FUNCTION_BLOCK FB_mF EXTENDS FB_StateSpaceModel
VAR_INPUT
END_VAR
VAR_OUTPUT
END_VAR
VAR
END_VAR

METHOD PUBLIC Init
VAR_INPUT
	activateObserver : BOOL;
END_VAR
VAR
    i,j : INT;
END_VAR

SUPER^();
nx := 2;
nu := 2;
ny := 1;

// Load matrices
_A[1,1] := 0.9895;
_A[1,2] := 0.03677;
_A[2,1] := -0.01237;
_A[2,2] := 0.9649;

_B[1,1] := -2.52E-05;
_B[1,2] := -1.673E-06;
_B[2,1] := -2.199E-04;
_B[2,2] := -5.346E-06;

_C[1,1] := -10.22;
_C[1,2] := -0.1235;

_K[1] := -0.1242;
_K[2] := -0.5091;
END_METHOD

END_FUNCTION_BLOCK

(* stored: Version 1.1.0.1, ProductVersion 3.1.4024.9
   POU FB_mF: Id {fbb14113-4232-402b-908d-7c31de6db086}, SpecialFunc None
   Method Init: Id {d3dfdef9-e2f9-4251-92e8-83806dad49e4} *)
